(* IEC 61131-3 sources: Lasal/CPU_5344_V01/Class/CanBase, 1 file *)

(* ---- CanBase.st ---- *)
(*!
<Class
	Name               = "CanBase"
	Revision           = "1.1"
	RealtimeTask       = "false"
	CyclicTask         = "true"
	BackgroundTask     = "false"
	Sigmatek           = "false"
	OSInterface        = "false"
	HighPriority       = "false"
	Automatic          = "false"
	UpdateMode         = "Prescan"
	SharedCommandTable = "true"
	Objectsize         = "(284,120)"
	Comment            = "CAN Base class">
	<Channels>
		<Server Name="Server0" Visualized="true" Initialize="false" WriteProtected="true" Retentive="false"/>
		<Client Name="Driver" Required="false" Internal="false"/>
		<Client Name="System" Required="false" Internal="false"/>
	</Channels>
	<Dependencies>
		<Files>
			<File Path=".\Class\CanBase\CanBaseGl.h" Include="false"/>
		</Files>
	</Dependencies>
	<RevDoku>
		<Owner Company="SigmaControl" Author="Johan Embregts"/>
		<Dokumentation Revision="1.1" Date="2013-06-20" Author="Johan Embregts" Company="SigmaControl" Description="ObjectClient Driver is not requiered."/>
	</RevDoku>
</Class>
*)
CanBase : CLASS
	TYPE
	  IntrStr : STRUCT  //! <Type Comment="Internal Class information" Name="IntrStr"/>
	    ObjInformation : LSLOBJ_INFO;  //! <Type Comment="Object information" Name="IntrStr.ObjInformation"/>
	  END_STRUCT;
	END_TYPE
  //Servers:
	Server0 	: SvrChCmd_DINT;
  //Clients:
	Driver 	: CltChCmd_CanDriverBase;
	System 	: CltChCmd_System;
  //Variables:
		Alive 	: DINT;			//! <Variable Comment="1= This station has been alive, 2= PollRequest" Name="Alive"/>
		tAlive 	: UDINT;			//! <Variable Comment="Time delay between keeping comm alive" Name="tAlive"/>
		tSend 	: UDINT;			//! <Variable Comment="Starttime send CAN object" Name="tSend"/>
		TxData 	: CanObjStr;			//! <Variable Comment="Send CAN object" Name="TxData"/>
		RxDataPtr 	: ^CanObjStr;			//! <Variable Comment="Recieve CAN object" Name="RxDataPtr"/>
		Intr 	: IntrStr;			//! <Variable Comment="Internal Class information" Name="Intr"/>
  //Functions:
				//! <Function Comment="[#ENGLISH]&#13;&#10;" Name="Init"/>
	FUNCTION VIRTUAL GLOBAL Init;
				//! <Function Comment="[#ENGLISH]&#13;&#10;" Name="CyWork"/>
	FUNCTION VIRTUAL GLOBAL CyWork
		VAR_INPUT
			EAX 	: UDINT := EAX;
		END_VAR
		VAR_OUTPUT
			state (EAX) 	: UDINT;
		END_VAR;
				//! <Function Comment=" 0 = OK.&#13;&#10;-1 = None existing CAN IO number.&#13;&#10;-2 = Size data buffer to Large.&#13;&#10;-3 = Driver client is not connected." Name="SendCanObj"/>
	FUNCTION VIRTUAL GLOBAL SendCanObj
		VAR_INPUT
			SendPtr 	: ^CanObjStr;			//! <Variable Comment="Pointer to CAN object to be send." Name="SendCanObj.SendPtr"/>
		END_VAR
		VAR_OUTPUT
			State 	: DINT;			//! <Variable Comment="0= ok, -1= ID error, -2= Size error." Name="SendCanObj.State"/>
		END_VAR;
				//! <Function Comment="[#ENGLISH]&#13;&#10;" Name="GetCanObj"/>
	FUNCTION VIRTUAL GLOBAL GetCanObj
		VAR_INPUT
			ObjNr 	: HDINT;			//! <Variable Comment="Test for a CAN Object with this ID." Name="GetCanObj.ObjNr"/>
		END_VAR
		VAR_OUTPUT
			Ptr2ID 	: ^CanObjStr;			//! <Variable Comment="Pointer to data of requested CAN object ID.&#13;&#10;When NIL no CAN object received or Client Driver not connected." Name="GetCanObj.Ptr2ID"/>
		END_VAR;
  //Tables:
	FUNCTION @STD
		VAR_OUTPUT
			ret_code	: CONFSTATES;
		END_VAR;
	FUNCTION GLOBAL TAB @CT_;
END_CLASS;

#pragma usingLtd CanDriverBase
#pragma usingLtd System

//*********************Inserted from .\CanBase\CanBase_00_00.st*********************

//[#ENGLISH]
(*	****************************************************************************************
	CANBase	driver to communicate with one CAN device
	****************************************************************************************

	Server	Server0		: 0				= Ok
						  -1			= Alive timeout.
	Client	Driver		: Connection to _CanDriverBase class for interface with the hardware
			System

	****************************************************************************************
	Created  : JE  : Wk 48/04	| Lasal V00:61f 	|
	Tested   : JE  : Wk 01/01	| Lasal V01:01:103	| c-IPC	- 2.2 x1.8	- 1.1.11 1.00.3.0
	Rev00:00 : JE  : Wk mm/yy	| Lasal Vxx:xxx		| c-IPC	-	-
	****************************************************************************************
//[#DEUTSCH]
(*	****************************************************************************************

	****************************************************************************************

	****************************************************************************************)

FUNCTION VIRTUAL GLOBAL CanBase::Init

(*
 * Synchronise timing with task.
 *)
System.GetObjectInfo( ThisObj0	:= This
					, TaskType0	:= Obj_Ct
					, ObjInfo	:= #Intr.ObjInformation);
(*
IF Intr.ObjInformation.OrgPeriod> 0 THEN
	TaskRes	:= to_dint( Intr.ObjInformation.OrgPeriod);	// this gives the ct timebase
ELSE
	Server0	:= -12;
END_IF;
*)
Alive	:= 0;

END_FUNCTION //VIRTUAL GLOBAL CanBase::Init

//[#ENGLISH]
(*	****************************************************************************************
	Cyclic task
	****************************************************************************************)

FUNCTION VIRTUAL GLOBAL CanBase::CyWork
VAR_INPUT
	EAX		: UDINT;
END_VAR
VAR_OUTPUT
	state		: UDINT;
END_VAR

// If no data within time recieved then device is not alive
If Alive> 0 Then
	If Ops.tAbsolute- tAlive> cCanOpenAliveTime Then
		Alive		:= 0;
	End_If;
End_If;

State	:= Ready$Dint;
END_FUNCTION //VIRTUAL GLOBAL CanBase::CyWork

//[#ENGLISH]
//[>ObjNr]Test for a CAN Object with this ID.
//[<Ptr2ID]Pointer to data of requested CAN object ID.
FUNCTION VIRTUAL GLOBAL CanBase::GetCanObj
VAR_INPUT
	ObjNr		: HDINT;
END_VAR
VAR_OUTPUT
	Ptr2ID		: ^CanObjStr;
END_VAR

if ObjNr <= cMaxCanMem
 & IsClientConnected( #Driver)
then
	Ptr2ID	:= Driver.GetObject( ObjNr);
	If Ptr2ID<> Nil Then
		Alive		:= 1;
		tAlive		:= Ops.tabsolute;
	End_If;
else
	Ptr2ID	:= Nil;
end_If;

END_FUNCTION //VIRTUAL GLOBAL CanBase::GetCanObj

//[#ENGLISH]
//[>SendPtr]Pointer to CAN object to be send.
//[<State]0= ok, -1= ID error, -2= Size error.
(*	****************************************************************************************
	Send a CAN object
	****************************************************************************************

	When the input object number "ObjNr" is recieved by the
	CAN Driver class then the return value will be the pointer
	to the recieved data in format "CanObjStr".
	the object number must be within the range of 0 and MaxCanMem_

	****************************************************************************************

	State	:  0	= ok.
			    -1	= None existing CAN ID number.
			    -2	= Size data bufer to large.
          -3  = Driver client is not connected.

	****************************************************************************************)
FUNCTION VIRTUAL GLOBAL CanBase::SendCanObj
VAR_INPUT
	SendPtr		: ^CanObjStr;
END_VAR
VAR_OUTPUT
	State		: DINT;
END_VAR

if IsClientConnected( #Driver) then
  if SendPtr^.ID<= cMaxCanMem then
    if SendPtr^.Size <= cMaxCanData then
      State	:= Driver.SendObject( TxBuffer	:= SendPtr);
      if State>= 0 then
        tSend	:= Ops.tAbsolute;
      end_if;
    else
      State	:= -2;
    end_If;
  else
    State	:= -1;
  end_if;
else
  State	:= -3;
end_if;

END_FUNCTION //VIRTUAL GLOBAL CanBase::SendCanObj
